(* IEC 61131-3 sources: industrial-ai-agent/templates/codesys/st-snippets, 7 files *)

(* ---- 05_opcua_symbol_publish.st ---- *)
// ============================================================
// OPC-UA Sembol Yayinlama Kaliplari
// Aciklama: PLC degiskenlerini OPC-UA'ya acmanin iki yolu:
//           (A) Symbol Configuration (UI'dan, kod gerekmez) - tavsiye edilen
//           (B) {attribute 'OPC.UA.DA' := '1'} pragma'lari ile kod icinde
//           Bu dosya pragma desenini, salt-okunur/yazilabilir ayrimini
//           ve HMI heartbeat (baglanti kopmasi tespiti) desenini gosterir.
// Altın kural: Kontrol mantigi HMI'da DEGIL PLC'de. HMI komut yazar,
//              PLC izin verirse uygular. Saldiri yuzeyini kucuk tut:
//              yalnizca gerekli degiskenleri ac.
// ============================================================

// ------------------------------------------------------------
// (A) Symbol Configuration yontemi (kod yok, ozet)
// ------------------------------------------------------------
// Application -> Add Object -> Symbol Configuration
//   [x] GVL_HMI_Read   -> Access Level: Read       (salt-okunur izleme)
//   [x] GVL_HMI_Cmd    -> Access Level: ReadWrite   (HMI komutlari)
// Build -> Download. NodeId formati:
//   ns=4;s=|var|<Runtime>.Application.GVL_HMI_Read.rSpeed
// NOT: Degisken adi = API sozlesmesi. Ad degisirse SCADA tag'i kopar.

// ============================================================
// GVL_HMI_Read - Salt-okunur izleme (PLC -> HMI)
// Pragma ile bu blok OPC-UA'ya read-only acilir.
// {attribute 'symbol' := 'read'} -> sembol seti erisimi read
// {attribute 'OPC.UA.DA' := '1'} -> node OPC-UA DA'da yayinlanir
// ============================================================
{attribute 'qualified_only'}
{attribute 'symbol' := 'read'}
VAR_GLOBAL
    {attribute 'OPC.UA.DA' := '1'}
    rSpeed        : REAL;           // m/min - olculen hiz (izleme)
    {attribute 'OPC.UA.DA' := '1'}
    rTemperature  : REAL;           // degC - sicaklik (izleme)
    {attribute 'OPC.UA.DA' := '1'}
    xRunning      : BOOL;           // Calisma durumu (izleme)
    {attribute 'OPC.UA.DA' := '1'}
    xAnyAlarm     : BOOL;           // Genel alarm ozeti (izleme)
    {attribute 'OPC.UA.DA' := '1'}
    nActiveAlarms : INT;            // Aktif alarm sayisi (izleme)
END_VAR

// ============================================================
// GVL_HMI_Cmd - Yazilabilir komutlar (HMI -> PLC)
// Bu degiskenler HMI'dan yazilir; PLC mantigi gecerliligini denetler.
// {attribute 'symbol' := 'readwrite'} -> okunur + yazilir
// ============================================================
{attribute 'qualified_only'}
{attribute 'symbol' := 'readwrite'}
VAR_GLOBAL
    {attribute 'OPC.UA.DA' := '1'}
    xCmdStart     : BOOL;           // HMI calistirma istegi (yalniz oto modda)
    {attribute 'OPC.UA.DA' := '1'}
    xCmdStop      : BOOL;           // HMI durdurma istegi
    {attribute 'OPC.UA.DA' := '1'}
    xCmdReset     : BOOL;           // HMI ariza sifirlama
    {attribute 'OPC.UA.DA' := '1'}
    rSetpoint     : REAL;           // HMI'dan setpoint (PLC kelepceler)
END_VAR

// ============================================================
// GVL_Heartbeat - HMI/SCADA baglanti gozlemi
// PLC her saniye uHbPlc'yi artirir; HMI bunu okuyup
// "PLC canli mi" anlar. HMI da uHbHmi'yi periyodik yazar;
// PLC bunu izleyip "HMI baglantisi kopdu mu" tespit eder.
// ============================================================
{attribute 'qualified_only'}
{attribute 'symbol' := 'readwrite'}
VAR_GLOBAL
    {attribute 'OPC.UA.DA' := '1'}
    uHbPlc        : UDINT;          // PLC -> HMI: PLC canlilik sayaci (read)
    {attribute 'OPC.UA.DA' := '1'}
    uHbHmi        : UDINT;          // HMI -> PLC: HMI canlilik sayaci (write)
    {attribute 'OPC.UA.DA' := '1'}
    xHmiConnected : BOOL;           // PLC tespiti: HMI baglantisi saglam mi
END_VAR

// ============================================================
// PRG_Heartbeat
// Aciklama: PLC heartbeat'i artirir ve HMI heartbeat'ini izler.
//           HMI uHbHmi'yi belirli surede degistirmezse baglanti
//           kopmus kabul edilir (xHmiConnected := FALSE).
//           Bu PROGRAM 100ms-1s araliginda bir task'ta cagrilmali.
// ============================================================
PROGRAM PRG_Heartbeat
VAR_INPUT
    tHmiTimeout   : TIME := T#5S;   // HMI bu surede degismezse kopuk say
    tPlcToggle    : TIME := T#1S;   // PLC heartbeat artirma periyodu
END_VAR
VAR
    tPlcTmr       : TON;
    tHmiTmr       : TON;
    uHbHmiPrev    : UDINT;
END_VAR

// --- PLC heartbeat: her tPlcToggle'da bir artir ---
tPlcTmr(IN := NOT tPlcTmr.Q, PT := tPlcToggle);
IF tPlcTmr.Q THEN
    GVL_Heartbeat.uHbPlc := GVL_Heartbeat.uHbPlc + 1;   // UDINT tasmasi normal (geri sarar)
END_IF

// --- HMI heartbeat izleme: degisiyor mu? ---
IF GVL_Heartbeat.uHbHmi <> uHbHmiPrev THEN
    // HMI heartbeat'i degisti -> baglanti canli, sayaci sifirla
    uHbHmiPrev := GVL_Heartbeat.uHbHmi;
    tHmiTmr(IN := FALSE);
    GVL_Heartbeat.xHmiConnected := TRUE;
ELSE
    // Degismedi -> zaman asimi say
    tHmiTmr(IN := TRUE, PT := tHmiTimeout);
    IF tHmiTmr.Q THEN
        GVL_Heartbeat.xHmiConnected := FALSE;   // HMI baglantisi koptu
    END_IF
END_IF

// Kullanim: baglanti kopunca HMI komutlarini yok say / guvenli duruma gec
// IF NOT GVL_Heartbeat.xHmiConnected THEN ... fail-safe ... END_IF

(* ---- 01_motor_start_stop.st ---- *)
// ============================================================
// FB_MotorStartStop
// Aciklama: Tek bir motorun start/stop mantigini yonetir.
//           Start butonu (NO), Stop butonu (NC tel-emniyetli),
//           interlock girisi, calisma geri beslemesi ve
//           kilitlenen (latch) ariza + reset icerir.
//           Tek sorumluluk: motor calistir/durdur mantigi.
//           Cikis I/O'ya YALNIZCA cagiran PROGRAM tarafindan baglanir.
// Not: Set/Reset cakismasinda STOP/ariza her zaman ONCELIKLIDIR
//      (reset dominant durdurma -> guvenli taraf).
// ============================================================
FUNCTION_BLOCK FB_MotorStartStop
VAR_INPUT
    // --- Komutlar ---
    xStartBtn   : BOOL;             // Start butonu (NO) - yukselen kenarda calistir
    xStopBtn    : BOOL;             // Stop butonu (NC) - TRUE = stop basili DEGIL
                                    //   yani kablo koparsa/buton basilirsa FALSE -> durdur
    xInterlock  : BOOL := TRUE;     // Calismaya izin (TRUE = izin var)
    xFaultReset : BOOL;             // Ariza sifirlama - yukselen kenar

    // --- Geri besleme ---
    xRunFeedback: BOOL;             // Kontaktor/yardimci kontak geri beslemesi

    // --- Konfigurasyon (sihirli sayi yok) ---
    tFbTimeout  : TIME := T#2S;     // Geri besleme gelmezse ariza gecikmesi
    bUseFeedback: BOOL := TRUE;     // FALSE -> geri besleme denetimi yapma
END_VAR
VAR_OUTPUT
    xRunOutput  : BOOL;             // Motor calistirma cikisi -> I/O'ya baglanir
    xRunning    : BOOL;             // Onaylanmis calisma durumu
    xReady      : BOOL;             // Bos, ariza yok, start bekliyor
    xFault      : BOOL;             // Kilitli ariza bayragi
    sFaultMsg   : STRING(80);       // Operatore bilgi mesaji
END_VAR
VAR
    fbStart     : R_TRIG;           // Start butonu yukselen kenar
    fbReset     : R_TRIG;           // Reset yukselen kenar
    tFbTimer    : TON;              // Geri besleme zaman asimi
    xCmdRun     : BOOL;             // Dahili calistirma istegi (latch)
END_VAR

// --- Kenar tespitleri (her scan cagrilmali) ---
fbStart(CLK := xStartBtn);
fbReset(CLK := xFaultReset);

// --- Ariza sifirlama (yalnizca kosul gitmisse) ---
IF fbReset.Q AND NOT (xRunFeedback AND NOT xRunOutput) THEN
    xFault    := FALSE;
    sFaultMsg := '';
END_IF

// --- Calistirma istegi: SET (start kenari) ---
IF fbStart.Q AND xInterlock AND NOT xFault THEN
    xCmdRun := TRUE;
END_IF

// --- Durdurma kosullari: RESET DOMINANT (guvenli taraf) ---
// Stop butonu NC: xStopBtn = FALSE -> durdur. Interlock kaybi -> durdur.
IF NOT xStopBtn OR NOT xInterlock OR xFault THEN
    xCmdRun := FALSE;
END_IF

// --- Fiziksel cikis ---
xRunOutput := xCmdRun AND NOT xFault;

// --- Geri besleme denetimi (kontaktor cekti mi?) ---
IF bUseFeedback THEN
    // Komut var ama geri besleme yok -> zaman asimi say
    tFbTimer(IN := (xRunOutput AND NOT xRunFeedback), PT := tFbTimeout);
    IF tFbTimer.Q THEN
        xFault    := TRUE;
        sFaultMsg := 'Motor calisma geri beslemesi yok. Kontaktor ve kabloyu kontrol edin.';
    END_IF

    // Komut yokken geri besleme varsa -> yapisik kontaktor (tehlikeli)
    IF NOT xRunOutput AND xRunFeedback THEN
        xFault    := TRUE;
        sFaultMsg := 'Beklenmeyen geri besleme. Kontaktor yapismis olabilir.';
    END_IF

    xRunning := xRunOutput AND xRunFeedback;
ELSE
    // Geri besleme yoksa cikis = calisma kabul edilir
    tFbTimer(IN := FALSE);
    xRunning := xRunOutput;
END_IF

// --- Hazir durumu ozeti ---
xReady := NOT xRunOutput AND NOT xFault AND xInterlock AND xStopBtn;

(* ---- 02_analog_scaling.st ---- *)
// ============================================================
// Analog Olcekleme Kalip Koleksiyonu
// Aciklama: FB_AnalogScale (ham -> muhendislik) projede mevcuttur
//           (projects/EXAMPLE_conveyor/program/03_FB_AnalogScale.st).
//           Bu dosya 3 ek kalip sunar:
//             1) FB_AnalogScale KULLANIM ornegi (cagri bicimi)
//             2) FB_EngToRaw  - tersine olcekleme (rEng -> iRaw, 4-20mA cikis)
//             3) FB_EMAFilter - ustel hareketli ortalama (gurultu filtresi)
// Not: Tum sabitler VAR_INPUT veya VAR CONSTANT; sifira bolme korumalidir.
// ============================================================

// ------------------------------------------------------------
// 1) KULLANIM ORNEGI - FB_AnalogScale + filtre zinciri
// ------------------------------------------------------------
// (Bir PROGRAM icinde tipik baglanti)
//
// VAR
//     fbScale  : FB_AnalogScale;
//     fbFilter : FB_EMAFilter;
//     rSpeed   : REAL;
// END_VAR
//
// fbScale(
//     iRaw      := GVL_IO.iSpeedRaw,   // Modul ham deger
//     iRawMin   := GVL_Const.RAW_4MA,
//     iRawMax   := GVL_Const.RAW_20MA,
//     rEngMin   := GVL_Const.SPEED_ENG_MIN,
//     rEngMax   := GVL_Const.SPEED_ENG_MAX,
//     iRawBreak := GVL_Const.RAW_BREAK
// );
//
// fbFilter(rIn := fbScale.rEng, rAlpha := 0.2);  // Yumusatma
// rSpeed := fbFilter.rOut;
//
// GVL_HMI.aZoneSpeed[1] := rSpeed;               // PROGRAM global'e yazar
// GVL_HMI.aZoneTacBrk[1] := fbScale.xUnderRange; // Kablo kopmasi

// ============================================================
// FB_EngToRaw
// Aciklama: Muhendislik birimini ham analog cikisa cevirir.
//           4-20mA analog cikis modulune deger gondermek icin.
//           FB_AnalogScale'in tersidir. Kelepceleme yapar.
// ============================================================
FUNCTION_BLOCK FB_EngToRaw
VAR_INPUT
    rEng     : REAL;    // Yazilacak muhendislik degeri (ornek: %valf acikligi)
    rEngMin  : REAL;    // Muhendislik min (4mA karsiligi)
    rEngMax  : REAL;    // Muhendislik max (20mA karsiligi)
    iRawMin  : INT;     // 4mA karsiligi ham deger
    iRawMax  : INT;     // 20mA karsiligi ham deger
END_VAR
VAR_OUTPUT
    iRaw     : INT;     // Module yazilacak ham deger
END_VAR
VAR
    rEngSpan : REAL;
    rClamped : REAL;
    rRaw     : REAL;
END_VAR

// --- Sifira bolme korumasi ---
rEngSpan := rEngMax - rEngMin;
IF rEngSpan = 0.0 THEN
    iRaw := iRawMin;          // Hatali konfig -> guvenli min cikis
    RETURN;
END_IF

// --- Giris kelepceleme (muhendislik araliginda tut) ---
rClamped := rEng;
IF rClamped > rEngMax THEN
    rClamped := rEngMax;
ELSIF rClamped < rEngMin THEN
    rClamped := rEngMin;
END_IF

// --- Tersine lineer olcekleme ---
rRaw := INT_TO_REAL(iRawMin) +
        ((rClamped - rEngMin) / rEngSpan) * INT_TO_REAL(iRawMax - iRawMin);

iRaw := REAL_TO_INT(rRaw);

// ============================================================
// FB_EMAFilter
// Aciklama: Ustel Hareketli Ortalama (EMA) ile analog sinyal
//           filtreleme. y = alpha*x + (1-alpha)*y_onceki.
//           alpha buyukse hizli (az filtre), kucukse yavas (cok filtre).
//           Gurultulu 4-20mA sinyallerini yumusatmak icin.
// ============================================================
FUNCTION_BLOCK FB_EMAFilter
VAR_INPUT
    rIn      : REAL;            // Ham (gurultulu) giris
    rAlpha   : REAL := 0.2;     // Filtre katsayisi (0.0 < alpha <= 1.0)
END_VAR
VAR_OUTPUT
    rOut     : REAL;            // Filtrelenmis cikis
END_VAR
VAR
    xFirst   : BOOL := TRUE;    // Ilk cevrimde dogrudan yukle
    rAlphaLim: REAL;
END_VAR

// --- Alpha sinir koruma (gecersiz deger filtreyi bozar) ---
rAlphaLim := rAlpha;
IF rAlphaLim <= 0.0 THEN
    rAlphaLim := 0.01;          // Cok yavas ama kararli
ELSIF rAlphaLim > 1.0 THEN
    rAlphaLim := 1.0;           // Filtre yok (cikis = giris)
END_IF

// --- Ilk cevrim: sicrama olmasin diye giris ile baslat ---
IF xFirst THEN
    rOut   := rIn;
    xFirst := FALSE;
ELSE
    rOut := rAlphaLim * rIn + (1.0 - rAlphaLim) * rOut;
END_IF

(* ---- 03_pid_loop.st ---- *)
// ============================================================
// FB_SimplePID
// Aciklama: Elle yazilmis konum-tipi (positional) PID kontrolor.
//           Anti-windup (integral clamp), manuel/oto bumpless
//           gecis ve cikis kelepceleme icerir.
//           Tek sorumluluk: PID hesabi (olcekleme/IO ayri FB'de).
// Not: CODESYS standart kutuphanesinde FB_PID hazir vardir;
//      bu FB egitim/tasinabilirlik icin saydam bir alternatiftir.
//      Her scan cagrilmali (TON yok ama integral durum tutar).
// Birim: rKp birimsiz; rTi/rTd SANIYE cinsinden; tCycle PID periyodu.
// ============================================================
FUNCTION_BLOCK FB_SimplePID
VAR_INPUT
    rActual    : REAL;              // Olcum (process value)
    rSetpoint  : REAL;              // Hedef deger

    // --- Mod ---
    bAuto      : BOOL := TRUE;      // FALSE -> manuel mod
    rManOut    : REAL;              // Manuel modda cikis degeri

    // --- PID parametreleri (sihirli sayi yok) ---
    rKp        : REAL := 1.0;       // Oransal kazanc
    rTi        : REAL := 10.0;      // Integral zamani [s] (0 = I kapali)
    rTd        : REAL := 0.0;       // Turev zamani [s]   (0 = D kapali)
    tCycle     : TIME := T#100MS;   // PID cevrim suresi (task cycle ile esit)

    // --- Cikis sinirlari ---
    rOutMin    : REAL := 0.0;       // Min cikis (ornek: %0)
    rOutMax    : REAL := 100.0;     // Max cikis (ornek: %100)
END_VAR
VAR_OUTPUT
    rOut       : REAL;              // PID cikisi (kelepcelenmis)
    bSatHigh   : BOOL;              // Cikis ust limitte (doygunluk)
    bSatLow    : BOOL;              // Cikis alt limitte (doygunluk)
    rError     : REAL;              // Anlik hata (SP - PV)
END_VAR
VAR
    rIntegral  : REAL;              // Integral birikim
    rPrevError : REAL;              // Onceki hata (turev icin)
    rDt        : REAL;              // Cevrim suresi [s]
    rP         : REAL;
    rI         : REAL;
    rD         : REAL;
    rRaw       : REAL;              // Kelepcelemeden onceki cikis
    bFirstScan : BOOL := TRUE;
END_VAR

// --- Cevrim suresi [s] (sifira bolme korumasi) ---
rDt := TIME_TO_REAL(tCycle) / 1000.0;
IF rDt <= 0.0 THEN
    rDt := 0.1;                     // Guvenli varsayilan 100ms
END_IF

// --- Limit tutarlilik korumasi ---
IF rOutMax <= rOutMin THEN
    rOutMax := rOutMin + 1.0;       // Hatali konfig -> en az 1 birim aralik
END_IF

rError := rSetpoint - rActual;

IF bAuto THEN
    // ---------- OTO MOD ----------
    // P terimi
    rP := rKp * rError;

    // I terimi (rTi=0 -> integral kapali)
    IF rTi > 0.0 THEN
        rIntegral := rIntegral + (rKp / rTi) * rError * rDt;
    ELSE
        rIntegral := 0.0;
    END_IF
    rI := rIntegral;

    // D terimi (turev; ilk scan'de atlama olmasin)
    IF (rTd > 0.0) AND NOT bFirstScan THEN
        rD := rKp * rTd * (rError - rPrevError) / rDt;
    ELSE
        rD := 0.0;
    END_IF

    rRaw := rP + rI + rD;

    // --- Cikis kelepceleme + ANTI-WINDUP ---
    // Cikis doygunlukta ise integrali geri sar (sinirda dondur).
    IF rRaw > rOutMax THEN
        rOut     := rOutMax;
        bSatHigh := TRUE;
        bSatLow  := FALSE;
        // Anti-windup: fazla biriken integrali geri al
        rIntegral := rIntegral - (rRaw - rOutMax);
    ELSIF rRaw < rOutMin THEN
        rOut     := rOutMin;
        bSatHigh := FALSE;
        bSatLow  := TRUE;
        rIntegral := rIntegral - (rRaw - rOutMin);
    ELSE
        rOut     := rRaw;
        bSatHigh := FALSE;
        bSatLow  := FALSE;
    END_IF

ELSE
    // ---------- MANUEL MOD ----------
    // Manuel cikisi kelepcele
    IF rManOut > rOutMax THEN
        rOut := rOutMax;
    ELSIF rManOut < rOutMin THEN
        rOut := rOutMin;
    ELSE
        rOut := rManOut;
    END_IF
    bSatHigh := FALSE;
    bSatLow  := FALSE;

    // BUMPLESS TRANSFER hazirligi:
    // Manueldeyken integrali mevcut cikisa esitle ki OTO'ya
    // gecince cikis sicramasin (P ve D anlik hesaplanir).
    rIntegral := rOut - rKp * rError;
END_IF

rPrevError := rError;
bFirstScan := FALSE;

// ------------------------------------------------------------
// CODESYS STANDART FB_PID KULLANIMI (alternatif)
// ------------------------------------------------------------
// VAR fbPID : FB_PID; END_VAR  // Standard.library / Util.library
//
// fbPID(
//     fActualValue   := rActual,
//     fSetpointValue := rSetpoint,
//     fKp            := 1.0,
//     fTn            := 10.0,                       // Integral zamani [s]
//     fTv            := 0.5,                        // Turev zamani [s]
//     fOutMinLimit   := 0.0,
//     fOutMaxLimit   := 100.0,
//     bManMode       := NOT bAuto,
//     fManValue      := rManOut,
//     fCycleTime     := TIME_TO_REAL(T#100MS) / 1000.0  // [s]
// );
// rOut := fbPID.fOut;

(* ---- 04_timer_patterns.st ---- *)
// ============================================================
// Timer Kalip Koleksiyonu (TON / TOF / TP)
// Aciklama: Endustride en sik kullanilan zamanlayici desenleri.
//           Tum TON/TOF/TP/BLINK bloklari HER SCAN cagrilmali;
//           kosullu cagri sayaci/zamani dondurur.
//           Sabitler VAR CONSTANT; sihirli sayi yok.
// Icindekiler:
//   1) FB_Debounce  - sinyal sicramasi temizleme (ornek: sikisma 200ms)
//   2) FB_OnDelay   - gecikmeli acma (delayed-on)
//   3) FB_Pulse     - tek atislik darbe (one-shot pulse)
//   4) FB_Blink     - lamba yanip sonme (blink/flash)
//   5) Retentive timer kalibi (akumulatif sure)
// ============================================================

// ============================================================
// FB_Debounce
// Aciklama: Gurultulu/sicrayan dijital girisi filtreler.
//           Giris stabil kalmadikca cikis degismez.
//           Ornek kullanim: sikisma sensoru 200ms debounce.
//           Hem yukselen hem dusen kenar icin ayri gecikme.
// ============================================================
FUNCTION_BLOCK FB_Debounce
VAR_INPUT
    xIn        : BOOL;              // Ham (gurultulu) giris
    tOnDelay   : TIME := T#200MS;   // Aktif kabul icin stabil kalma suresi
    tOffDelay  : TIME := T#200MS;   // Pasif kabul icin stabil kalma suresi
END_VAR
VAR_OUTPUT
    xOut       : BOOL;              // Filtrelenmis (debounce edilmis) cikis
    xRising    : BOOL;              // Cikista yukselen kenar (tek scan)
    xFalling   : BOOL;              // Cikista dusen kenar (tek scan)
END_VAR
VAR
    tOn        : TON;
    tOff       : TON;
    xOutPrev   : BOOL;
END_VAR

// Giris TRUE'da kalmissa onu kabul et
tOn(IN := xIn, PT := tOnDelay);
// Giris FALSE'ta kalmissa onu kabul et
tOff(IN := NOT xIn, PT := tOffDelay);

IF tOn.Q THEN
    xOut := TRUE;
ELSIF tOff.Q THEN
    xOut := FALSE;
END_IF

xRising  := xOut AND NOT xOutPrev;
xFalling := NOT xOut AND xOutPrev;
xOutPrev := xOut;

// ============================================================
// FB_OnDelay
// Aciklama: Giris TRUE olduktan tPreset sure sonra cikis TRUE.
//           Giris FALSE olunca cikis aninda FALSE (klasik TON).
//           Ornek: motor calistiktan 3s sonra "kararli" bayragi.
// ============================================================
FUNCTION_BLOCK FB_OnDelay
VAR_INPUT
    xIn        : BOOL;
    tPreset    : TIME := T#3S;      // Gecikme suresi
END_VAR
VAR_OUTPUT
    xOut       : BOOL;              // Gecikmeli cikis
    tElapsed   : TIME;              // Gecen sure (HMI gosterimi)
END_VAR
VAR
    tDelay     : TON;
END_VAR

tDelay(IN := xIn, PT := tPreset);
xOut     := tDelay.Q;
tElapsed := tDelay.ET;

// ============================================================
// FB_Pulse
// Aciklama: Yukselen kenarda sabit sureli tek darbe uretir (TP).
//           Giris ne kadar uzun TRUE kalirsa kalsin darbe suresi sabit.
//           Ornek: buton basisinda 500ms'lik sesli uyari/kornaya darbe.
// ============================================================
FUNCTION_BLOCK FB_Pulse
VAR_INPUT
    xTrig      : BOOL;              // Tetik (yukselen kenar)
    tWidth     : TIME := T#500MS;   // Darbe genisligi
END_VAR
VAR_OUTPUT
    xPulse     : BOOL;              // Darbe cikisi
END_VAR
VAR
    fbTP       : TP;
END_VAR

fbTP(IN := xTrig, PT := tWidth);
xPulse := fbTP.Q;

// ============================================================
// FB_Blink
// Aciklama: Cikisi simetrik/asimetrik yanip-sondurur (lamba flash).
//           xEnable TRUE iken tOn/tOff periyotlariyla titresir.
//           Ornek: aktif alarm lambasi yanip sonsun.
// ============================================================
FUNCTION_BLOCK FB_Blink
VAR_INPUT
    xEnable    : BOOL;              // Yanip sonmeyi etkinlestir
    tOnTime    : TIME := T#500MS;   // Yanik kalma suresi
    tOffTime   : TIME := T#500MS;   // Sonuk kalma suresi
END_VAR
VAR_OUTPUT
    xOut       : BOOL;              // Lamba cikisi
END_VAR
VAR
    tOnTmr     : TON;
    tOffTmr    : TON;
END_VAR

IF NOT xEnable THEN
    xOut := FALSE;
    tOnTmr(IN := FALSE);
    tOffTmr(IN := FALSE);
ELSE
    // Sonuk fazi bitince yak; yanik fazi bitince sondur
    tOffTmr(IN := NOT xOut, PT := tOffTime);
    IF tOffTmr.Q THEN
        xOut := TRUE;
    END_IF

    tOnTmr(IN := xOut, PT := tOnTime);
    IF tOnTmr.Q THEN
        xOut := FALSE;
    END_IF
END_IF

// ============================================================
// FB_RetentiveTimer
// Aciklama: Akumulatif (retentive) zamanlayici. TON'dan farki:
//           giris kesilince sayac SIFIRLANMAZ, durur ve kaldigi
//           yerden devam eder. xReset ile sifirlanir.
//           Ornek: motorun toplam calisma suresini olcmek.
// ============================================================
FUNCTION_BLOCK FB_RetentiveTimer
VAR_INPUT
    xIn        : BOOL;              // Sayma kosulu (TRUE iken biriktir)
    xReset     : BOOL;              // Akumlatoru sifirla
    tPreset    : TIME := T#0S;      // 0 = sinir yok; >0 ise Q icin esik
END_VAR
VAR_OUTPUT
    tAccum     : TIME;              // Birikmis sure
    xDone      : BOOL;              // tAccum >= tPreset (preset>0 ise)
END_VAR
VAR
    tSlice     : TON;               // Bir scan'lik dilim olcumu
    tCycle     : TIME := T#10MS;    // Task cycle time (gercege gore ayarla)
END_VAR

IF xReset THEN
    tAccum := T#0S;
    xDone  := FALSE;
END_IF

// Her scan, kosul aktifse cycle time kadar ekle
IF xIn THEN
    tAccum := tAccum + tCycle;
END_IF

IF tPreset > T#0S THEN
    xDone := tAccum >= tPreset;
END_IF

(* ---- 06_alarm_handling.st ---- *)
// ============================================================
// Alarm Yonetimi Kaliplari
// Aciklama: Alarm latch (gelme/gitme/kabul), seviye siniflandirma,
//           zaman damgasi ve aktif alarm sayaci icerir.
//           Tek alarm noktasi -> FB_Alarm; toplu yonetim -> PRG_AlarmManager.
// Onemli: Analog tetikli alarmlara histerezis + debounce ekleyin
//         (alarm chattering / sel baskini onleme).
// ============================================================

// ------------------------------------------------------------
// Alarm seviyesi (DUT dosyasinda tanimlanir)
// ------------------------------------------------------------
// TYPE E_AlarmLevel :
// (
//     eLevel_None     := 0,
//     eLevel_Dusuk    := 1,   // Bilgi - makine durmaz
//     eLevel_Orta     := 2,   // Uyari - dikkat
//     eLevel_Yuksek   := 3,   // Onemli - mudahale gerek
//     eLevel_Kritik   := 4    // Makine durmali
// );
// END_TYPE

// ============================================================
// FB_Alarm
// Aciklama: Tek bir alarm noktasini yonetir. Latch davranisli:
//           tetik gelince aktif olur, kosul gitse bile operator
//           kabul edene (Ack) kadar kayitli kalir.
//           Yasam dongusu: Gelme -> (Ack) -> Gitme -> Temizlenme.
// Tek sorumluluk: bir alarmin durum makinesi.
// ============================================================
FUNCTION_BLOCK FB_Alarm
VAR_INPUT
    xTrigger    : BOOL;             // Alarm kosulu (TRUE = aktif olmali)
    xAckCmd     : BOOL;             // Operator kabul komutu (yukselen kenar)
    eLevel      : E_AlarmLevel := eLevel_Orta;  // Alarm seviyesi
    sMessage    : STRING(80) := '';             // Operator mesaji
END_VAR
VAR_OUTPUT
    xActive     : BOOL;             // Alarm halen aktif (kosul var)
    xLatched    : BOOL;             // Kayitli (aktif veya kabul bekliyor)
    xUnacked    : BOOL;             // Aktif ama kabul edilmedi (yanip sonme icin)
    dtOnset     : DATE_AND_TIME;    // Geldigi an (zaman damgasi)
    dtClear     : DATE_AND_TIME;    // Gittigi an (zaman damgasi)
END_VAR
VAR
    fbOn        : R_TRIG;           // Tetik yukselen kenar (gelme)
    fbOff       : F_TRIG;           // Tetik dusen kenar (gitme)
    fbAck       : R_TRIG;           // Kabul yukselen kenar
    xAcked      : BOOL;             // Kabul edildi mi
END_VAR

fbOn(CLK := xTrigger);
fbOff(CLK := xTrigger);
fbAck(CLK := xAckCmd);

// --- GELME: yeni alarm ---
IF fbOn.Q THEN
    xLatched := TRUE;
    xAcked   := FALSE;
    dtOnset  := NOW();              // NOT: RTC pili bitikse zaman damgasi bozulur
END_IF

// --- GITME: kosul ortadan kalkti ---
IF fbOff.Q THEN
    dtClear := NOW();
END_IF

// --- KABUL: operator onayladi ---
IF fbAck.Q AND xLatched THEN
    xAcked := TRUE;
END_IF

// --- TEMIZLENME: kosul gitti VE kabul edildi ---
IF NOT xTrigger AND xAcked THEN
    xLatched := FALSE;
END_IF

// --- Cikis ozetleri ---
xActive  := xTrigger;
xUnacked := xLatched AND NOT xAcked;

// ============================================================
// FB_AnalogAlarm
// Aciklama: Analog deger esik asimi alarmi. HISTEREZIS (set != reset)
//           ve DEBOUNCE (TON) ile chattering onler.
//           Ornek: sicaklik > 80 -> alarm; < 78 -> temizle.
// ============================================================
FUNCTION_BLOCK FB_AnalogAlarm
VAR_INPUT
    rValue      : REAL;             // Izlenen deger
    rSetLimit   : REAL := 80.0;     // Alarm tetik esigi
    rResetLimit : REAL := 78.0;     // Alarm cikis esigi (histerezis bandi)
    tDebounce   : TIME := T#500MS;  // Esik asimi stabil kalma suresi
    bHighAlarm  : BOOL := TRUE;     // TRUE=yuksek alarm, FALSE=dusuk alarm
END_VAR
VAR_OUTPUT
    xAlarm      : BOOL;             // Debounce'li alarm cikisi
END_VAR
VAR
    xRaw        : BOOL;             // Histerezisli ham alarm
    tDeb        : TON;
END_VAR

// --- Histerezis (Schmitt-trigger): yon'e gore esikler ---
IF bHighAlarm THEN
    IF rValue >= rSetLimit THEN
        xRaw := TRUE;
    ELSIF rValue <= rResetLimit THEN
        xRaw := FALSE;
    END_IF
ELSE
    // Dusuk alarm: deger esik altina dusunce tetik
    IF rValue <= rSetLimit THEN
        xRaw := TRUE;
    ELSIF rValue >= rResetLimit THEN
        xRaw := FALSE;
    END_IF
END_IF

// --- Debounce: kisa sicramalari yut ---
tDeb(IN := xRaw, PT := tDebounce);
xAlarm := tDeb.Q;

// ============================================================
// PRG_AlarmManager
// Aciklama: Birden cok FB_Alarm instance'ini yonetir, aktif
//           alarm sayisini ve seviye ozetlerini hesaplar.
//           Tum alarm degerlendirmesi orta hizli (10-50ms) task'ta.
// ============================================================
PROGRAM PRG_AlarmManager
VAR
    afbAlarm      : ARRAY[1..16] OF FB_Alarm;   // 16 alarm noktasi
    nActiveCount  : INT;                        // Aktif alarm sayisi
    nUnackedCount : INT;                        // Kabul edilmemis sayisi
    xAnyCritical  : BOOL;                       // Kritik alarm var mi
    xAnyAlarm     : BOOL;                       // Herhangi alarm var mi
    i             : INT;
END_VAR

// --- Ornek: 1 ve 2 numarali alarmlari besle (digerleri benzer) ---
afbAlarm[1](
    xTrigger := GVL_IO.xEStop,
    xAckCmd  := GVL_HMI_Cmd.xCmdReset,
    eLevel   := eLevel_Kritik,
    sMessage := 'Acil stop basili. Reset icin kurtarip onaylayin.'
);
afbAlarm[2](
    xTrigger := GVL_IO.xMotor1Fault,
    xAckCmd  := GVL_HMI_Cmd.xCmdReset,
    eLevel   := eLevel_Yuksek,
    sMessage := 'Motor 1 ariza. Kontaktor K1 kontrol edin.'
);

// --- Ozet sayaclari sifirla, sonra dongude topla ---
nActiveCount  := 0;
nUnackedCount := 0;
xAnyCritical  := FALSE;

FOR i := 1 TO 16 DO
    IF afbAlarm[i].xActive THEN
        nActiveCount := nActiveCount + 1;
        IF afbAlarm[i].eLevel = eLevel_Kritik THEN
            xAnyCritical := TRUE;
        END_IF
    END_IF
    IF afbAlarm[i].xUnacked THEN
        nUnackedCount := nUnackedCount + 1;
    END_IF
END_FOR

xAnyAlarm := nActiveCount > 0;

// --- Global izleme degiskenlerine aktar (PROGRAM yazar) ---
GVL_HMI_Read.nActiveAlarms := nActiveCount;
GVL_HMI_Read.xAnyAlarm     := xAnyAlarm;

(* ---- 07_error_watchdog.st ---- *)
// ============================================================
// Hata Yonetimi ve Watchdog Kaliplari
// Aciklama: Haberlesme/HMI watchdog (heartbeat timeout), task
//           watchdog kavrami, guvenli duruma gecis (fail-safe)
//           ve TRY benzeri hata yonetimi (CmpError/status kodu).
// Hata yonetimi felsefesi (knowledge/.../05_error_handling.md):
//   Savunmaci onleme + katmanli fail-safe. CODESYS'te genel
//   try/catch yoktur (64-bit'te __TRY hic yok). Onleme esastir.
// ============================================================

// ============================================================
// FB_CommWatchdog
// Aciklama: Bir haberlesme/HMI ortaginin heartbeat'ini izler.
//           Sayac belirli surede degismezse "kopuk" tespit eder.
//           Toparlanma: sayac yeniden degisirse otomatik temizlenir.
// Tek sorumluluk: heartbeat zaman asimi tespiti.
// ============================================================
FUNCTION_BLOCK FB_CommWatchdog
VAR_INPUT
    uHeartbeat  : UDINT;            // Karsi tarafin canlilik sayaci
    tTimeout    : TIME := T#3S;     // Bu surede degismezse kopuk say
    xEnable     : BOOL := TRUE;     // FALSE -> izleme yapma (saglikli kabul)
END_VAR
VAR_OUTPUT
    xConnected  : BOOL := TRUE;     // Baglanti saglam mi
    xTimeout    : BOOL;             // Zaman asimi olustu mu
    uFailCount  : UDINT;            // Toplam kopma sayisi (diagnostik)
END_VAR
VAR
    uHbPrev     : UDINT;
    tWdTmr      : TON;
    xWasConn    : BOOL := TRUE;
END_VAR

IF NOT xEnable THEN
    xConnected := TRUE;
    xTimeout   := FALSE;
    tWdTmr(IN := FALSE);
    uHbPrev    := uHeartbeat;
    RETURN;
END_IF

IF uHeartbeat <> uHbPrev THEN
    // Heartbeat ilerledi -> baglanti canli
    uHbPrev := uHeartbeat;
    tWdTmr(IN := FALSE);
    xConnected := TRUE;
    xTimeout   := FALSE;
ELSE
    // Degismedi -> zaman asimi say
    tWdTmr(IN := TRUE, PT := tTimeout);
    IF tWdTmr.Q THEN
        xConnected := FALSE;
        xTimeout   := TRUE;
    END_IF
END_IF

// Yeni kopma kenarini say (diagnostik)
IF xWasConn AND NOT xConnected THEN
    uFailCount := uFailCount + 1;
END_IF
xWasConn := xConnected;

// ============================================================
// FB_TryReadStatus - TRY benzeri durum-kodu hata yonetimi
// Aciklama: CODESYS'te genel try/catch yerine kutuphane FB'leri
//           bir status/error kodu doner (CmpError mantigi).
//           Bu sablon o kodu yorumlayip katmanli tepki uretir:
//           yeniden dene -> belirli sayidan sonra ariza.
// Not: 64-bit sistemde __TRY/__CATCH calismaz; savunmaci
//      durum-kodu denetimi tasinabilir ve guvenli yoldur.
// ============================================================
FUNCTION_BLOCK FB_TryReadStatus
VAR_INPUT
    xDone       : BOOL;             // Islem tamamlandi (kutuphane FB cikisi)
    xError      : BOOL;             // Islem hatali (kutuphane FB cikisi)
    wErrorId    : WORD;             // Hata kodu (kutuphane FB cikisi)
    nMaxRetries : INT := 3;         // Ariza ilan etmeden once deneme sayisi
    tRetryDelay : TIME := T#1S;     // Denemeler arasi bekleme
END_VAR
VAR_OUTPUT
    xOk         : BOOL;             // Basariyla tamamlandi
    xRetry      : BOOL;             // Yeniden deneme tetigi (tek scan)
    xFault      : BOOL;             // Kalici ariza (deneme tukendi)
    nRetryCount : INT;              // Yapilan deneme sayisi
    sFaultMsg   : STRING(80);
END_VAR
VAR
    fbErr       : R_TRIG;
    tRetryTmr   : TON;
END_VAR

xRetry := FALSE;
fbErr(CLK := xError);

IF xDone AND NOT xError THEN
    // --- Basari: temizle ---
    xOk         := TRUE;
    xFault      := FALSE;
    nRetryCount := 0;
    sFaultMsg   := '';
    tRetryTmr(IN := FALSE);

ELSIF fbErr.Q THEN
    // --- Yeni hata kenari: say ---
    xOk := FALSE;
    nRetryCount := nRetryCount + 1;

    IF nRetryCount >= nMaxRetries THEN
        // Deneme tukendi -> kalici ariza
        xFault    := TRUE;
        sFaultMsg := CONCAT('Islem basarisiz. Hata kodu: ', WORD_TO_STRING(wErrorId));
    ELSE
        // Yeniden denemek icin bekleme baslat
        tRetryTmr(IN := TRUE, PT := tRetryDelay);
    END_IF

ELSIF tRetryTmr.Q THEN
    // --- Bekleme bitti -> yeniden dene ---
    tRetryTmr(IN := FALSE);
    xRetry := TRUE;
END_IF

// ============================================================
// PRG_SafeState - Fail-safe (guvenli duruma gecis)
// Aciklama: Kritik hata/watchdog/baglanti kopmasi durumunda
//           tum tehlikeli ciktilari guvenli konuma getirir.
//           IDEAL: ayri, yuksek oncelikli Task_Safety'de calistir;
//           boylece Task_Control watchdog'undan bagimsiz korur.
// UYARI: CODESYS V3'te watchdog SADECE application'i durdurur;
//        fiziksel cikislar fieldbus fail-safe ayarina gore davranir
//        (otomatik 0 DEGIL). Slave fail-safe degerleri ayrica
//        konfigure edilmeli ve fiziksel test edilmelidir.
// ============================================================
PROGRAM PRG_SafeState
VAR_INPUT
    xSystemOk     : BOOL;           // Genel sistem saglikli mi
    xCommOk       : BOOL;           // Haberlesme saglikli mi
    xAnyCritical  : BOOL;           // Kritik alarm var mi
END_VAR
VAR
    xSafeStateNeeded : BOOL;
END_VAR

// --- Guvenli durum kosulu ---
xSafeStateNeeded := NOT xSystemOk OR NOT xCommOk OR xAnyCritical;

IF xSafeStateNeeded THEN
    // Tum tehlikeli ciktilari kapat (fail-safe)
    GVL_IO.xMotor1Out := FALSE;
    GVL_IO.xMotor2Out := FALSE;
    GVL_IO.xHeaterOut := FALSE;
    GVL_IO.xValveOut  := FALSE;     // NOT: vana fail-safe yonu prosese gore
END_IF

// ============================================================
// Task Watchdog yapilandirmasi (kavram - kod degil)
// ============================================================
// Task Configuration -> MainTask -> Configuration:
//   Watchdog        : Enabled
//   Time            : ~2-5 x beklenen Max Exec Time (ornek t#50ms)
//   Sensitivity     : 2-3 (tek spike'i tolere et, kalici sorunu yakala)
//
// Watchdog tetiklenince (V3):
//   1. Etkilenen Application durur (runtime devam eder)
//   2. Fiziksel cikislar -> fieldbus fail-safe ayarina gore
//   3. CODESYS Log'a kayit
//   4. Otomatik restart YOK - Application event handler gerekir
//
// Guvenlik: kritik cikislari ayri Task_Safety + donanim watchdog
//           rolesi ile koru. "STOP = guvenli" otomatik DEGILDIR.
